PROGRAM MAIN
VAR
	x : INT;
END_VAR

IF x < 100 THEN
	x := x+1;
END_IF

END_PROGRAM

(* stored: Version 1.1.0.1, ProductVersion 3.1.4024.2
   POU MAIN: Id {86704359-087c-4339-a0ee-37cc917d210f}, SpecialFunc None *)
